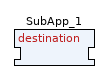
      [picture p49: application EventConnectionTestApp.Test14]
      SUBAPPLICATION SubApp_1
        EVENT_INPUT
          destination;
        END_EVENT
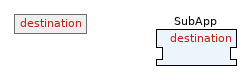
        SUBAPPLICATION SubApp
          EVENT_OUTPUT
            destination;
          END_EVENT
        END_SUBAPPLICATION
      END_SUBAPPLICATION
    END_SUBAPPLICATION
    SUBAPPLICATION SubApp_10
      EVENT_INPUT
        source;
      END_EVENT
    END_SUBAPPLICATION
    SUBAPPLICATION SubApp_11
      EVENT_INPUT
        source;
      END_EVENT
    END_SUBAPPLICATION
    SUBAPPLICATION Test14Solution
      EVENT_OUTPUT
        destination;
      END_EVENT
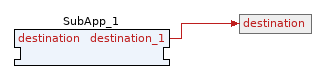
      SUBAPPLICATION SubApp_1
        EVENT_INPUT
          destination;
        END_EVENT
        EVENT_OUTPUT
          destination_1;
        END_EVENT
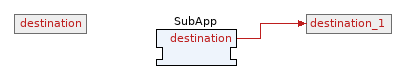
        SUBAPPLICATION SubApp
          EVENT_OUTPUT
            destination;
          END_EVENT
        END_SUBAPPLICATION
        EVENT_CONNECTIONS
          SubApp.destination TO destination_1;
        END_CONNECTIONS
      END_SUBAPPLICATION
      EVENT_CONNECTIONS
        SubApp_1.destination_1 TO destination;
      END_CONNECTIONS
    END_SUBAPPLICATION
    SUBAPPLICATION Test15 (* event input already exists inwards *)
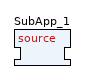
      SUBAPPLICATION SubApp_1
        EVENT_INPUT
          source;
        END_EVENT
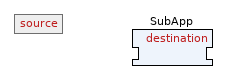
        SUBAPPLICATION SubApp
          EVENT_OUTPUT
            destination;
          END_EVENT
        END_SUBAPPLICATION
      END_SUBAPPLICATION
    END_SUBAPPLICATION
    SUBAPPLICATION SubApp_12
      EVENT_OUTPUT
        source;
      END_EVENT
    END_SUBAPPLICATION
    SUBAPPLICATION SubApp_13
      EVENT_OUTPUT
        source;
      END_EVENT
    END_SUBAPPLICATION
    SUBAPPLICATION Test15Solution
      EVENT_INPUT
        source;
      END_EVENT
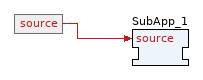
      SUBAPPLICATION SubApp_1
        EVENT_INPUT
          source;
        END_EVENT
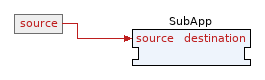
        SUBAPPLICATION SubApp
          EVENT_INPUT
            source;
          END_EVENT
          EVENT_OUTPUT
            destination;
          END_EVENT
          EVENT_CONNECTIONS
            source TO destination;
          END_CONNECTIONS
        END_SUBAPPLICATION
        EVENT_CONNECTIONS
          source TO SubApp.source;
        END_CONNECTIONS
      END_SUBAPPLICATION
      EVENT_CONNECTIONS
        source TO SubApp_1.source;
      END_CONNECTIONS
    END_SUBAPPLICATION
    SUBAPPLICATION Test16 (* event input pin with same name already exists, inwards *)
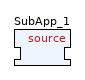
      SUBAPPLICATION SubApp_1
        EVENT_OUTPUT
          source;
        END_EVENT
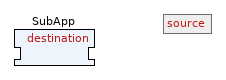
        SUBAPPLICATION SubApp
          EVENT_OUTPUT
            destination;
          END_EVENT
        END_SUBAPPLICATION
      END_SUBAPPLICATION
    END_SUBAPPLICATION
    SUBAPPLICATION SubApp_14
      EVENT_OUTPUT
        source;
      END_EVENT
    END_SUBAPPLICATION
    SUBAPPLICATION Test16Solution
      EVENT_INPUT
        source;
      END_EVENT
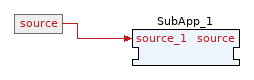
      SUBAPPLICATION SubApp_1
        EVENT_INPUT
          source_1;
        END_EVENT
        EVENT_OUTPUT
          source;
        END_EVENT
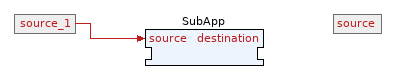
        SUBAPPLICATION SubApp
          EVENT_INPUT
            source;
          END_EVENT
          EVENT_OUTPUT
            destination;
          END_EVENT
          EVENT_CONNECTIONS
            source TO destination;
          END_CONNECTIONS
        END_SUBAPPLICATION
        EVENT_CONNECTIONS
          source_1 TO SubApp.source;
        END_CONNECTIONS
      END_SUBAPPLICATION
      EVENT_CONNECTIONS
        source TO SubApp_1.source_1;
      END_CONNECTIONS
    END_SUBAPPLICATION
    SUBAPPLICATION SubApp_15
      EVENT_OUTPUT
        source;
      END_EVENT
    END_SUBAPPLICATION
    SUBAPPLICATION Test17 (* interface to interface across hierarchies, swap *)
      EVENT_OUTPUT
        source;
      END_EVENT
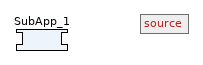
      SUBAPPLICATION SubApp_1
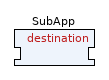
        SUBAPPLICATION SubApp
          EVENT_OUTPUT
            destination;
          END_EVENT
        END_SUBAPPLICATION
      END_SUBAPPLICATION
    END_SUBAPPLICATION
    SUBAPPLICATION Test18 (* interface to interface across hierarchies, no swap *)
      EVENT_OUTPUT
        destination;
      END_EVENT
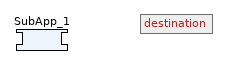
      SUBAPPLICATION SubApp_1
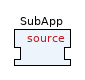
        SUBAPPLICATION SubApp
          EVENT_OUTPUT
            source;
          END_EVENT
        END_SUBAPPLICATION
      END_SUBAPPLICATION
    END_SUBAPPLICATION
    SUBAPPLICATION Test19
      EVENT_INPUT
        source;
      END_EVENT
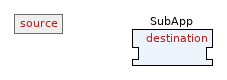
      SUBAPPLICATION SubApp
        EVENT_OUTPUT
          destination;
        END_EVENT
      END_SUBAPPLICATION
    END_SUBAPPLICATION
    SUBAPPLICATION Test20
      EVENT_INPUT
        destination;
      END_EVENT
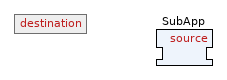
      SUBAPPLICATION SubApp
        EVENT_OUTPUT
          source;
        END_EVENT
      END_SUBAPPLICATION
    END_SUBAPPLICATION
    SUBAPPLICATION Test21
      EVENT_OUTPUT
        destination;
      END_EVENT
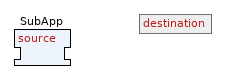
      SUBAPPLICATION SubApp
        EVENT_INPUT
          source;
        END_EVENT
      END_SUBAPPLICATION
    END_SUBAPPLICATION
    EVENT_CONNECTIONS
      fb_destinationevent_1.destination TO Test4Solution.destination;
      Test5Solution.destination TO fb_destinationevent_3.source;
      Test6Solution.destination TO fb_destinationevent_5.source;
      Test7Solution.destination TO fb_destinationevent_7.source;
      SubApp_1.destination TO Test9Solution.destination;
      SubApp_3.source TO Test10Solution.source;
      SubApp_5.source TO Test11Solution.source;
      Test12Solution.destination TO SubApp_7.source;
      Test13Solution.destination TO SubApp_9.source;
      Test14Solution.destination TO SubApp_11.source;
      SubApp_13.source TO Test15Solution.source;
      SubApp_15.source TO Test16Solution.source;
    END_CONNECTIONS
  END_APPLICATION
  APPLICATION DataConnectionTestApp
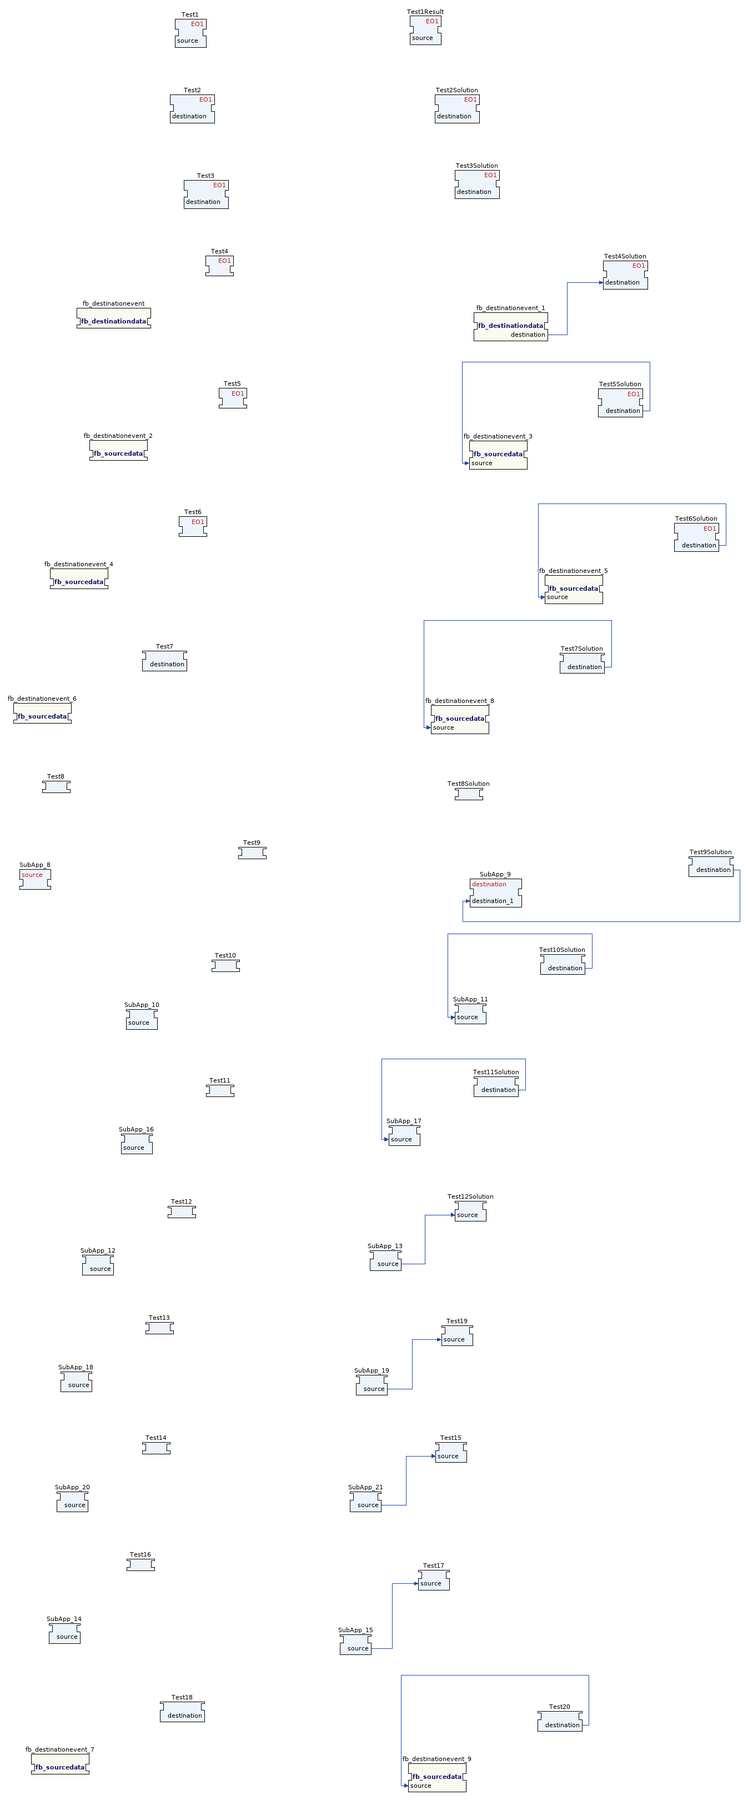
    FBS
      fb_destinationevent : fb_destinationdata;
      fb_destinationevent_1 : fb_destinationdata;
      fb_destinationevent_2 : fb_sourcedata;
      fb_destinationevent_3 : fb_sourcedata;
      fb_destinationevent_4 : fb_sourcedata;
      fb_destinationevent_5 : fb_sourcedata;
      fb_destinationevent_6 : fb_sourcedata;
      fb_destinationevent_7 : fb_sourcedata;
      fb_destinationevent_8 : fb_sourcedata;
      fb_destinationevent_9 : fb_sourcedata;
    END_FBS
    SUBAPPLICATION Test1 (* connection between subapp borders *)
      EVENT_OUTPUT
        EO1;
      END_EVENT
      VAR_INPUT
        source : BOOL;
      END_VAR
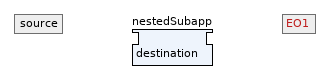
      SUBAPPLICATION nestedSubapp
        VAR_INPUT
          destination : BOOL;
        END_VAR
      END_SUBAPPLICATION
    END_SUBAPPLICATION
    SUBAPPLICATION Test3 (* crossing connection from FB to subapp border *)
      EVENT_OUTPUT
        EO1;
      END_EVENT
      VAR_INPUT
        destination : BOOL;
      END_VAR
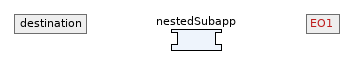
      SUBAPPLICATION nestedSubapp
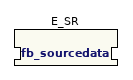
        FBS
          E_SR : fb_sourcedata;
        END_FBS
      END_SUBAPPLICATION
    END_SUBAPPLICATION
    SUBAPPLICATION Test4 (* crossing connection from FB in nested subapp to FB via app network *)
      EVENT_OUTPUT
        EO1;
      END_EVENT
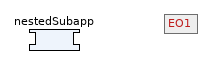
      SUBAPPLICATION nestedSubapp
